// TIA Portal V17 export
// export: Created 2024-08-26T21:07:14.5567643Z, ExportSetting WithDefaults, DisplayName Totally Integrated Automation Portal, DisplayVersion V17 Update 7, DisplayName TIA Portal Openness, DisplayVersion V17 Update 7, DisplayName TIA Portal Version Control Interface, DisplayVersion V17, DisplayName SINAMICS Startdrive Advanced, DisplayVersion V17 SP2, DisplayName SINAMICS Startdrive G110M, G120, G120C, G120D, G120P, G115D, DisplayVersion V17 SP2, DisplayName SINAMICS Startdrive G130, G150, S120, S150, SINAMICS MV, S210, DisplayVersion V17 SP2, DisplayName STEP 7 Professional, DisplayVersion V17 Update 7, DisplayName STEP 7 Safety, DisplayVersion V17 Update 6, DisplayName WinCC Advanced / Unified PC, DisplayVersion V17 Update 7
ORGANIZATION_BLOCK "Main"   // OB1, LAD, ProgramCycle
TITLE = "Main Program Sweep (Cycle)"
{ S7_Optimized_Access := 'TRUE' }
VERSION : 0.1
// stored: AutoNumber true, IsIECCheckEnabled false, SetENOAutomatically false
   VAR_INPUT
      Initial_Call : Bool;   // Initial call of this OB
      Remanence : Bool;   // =True, if remanent data are available
   END_VAR
   VAR_TEMP
      BUFFER : String;
   END_VAR
   VAR_TEMP   // added for the SCL form of the ladder/FBD networks
      _w1 : Bool;
      _w2 : Bool;
      _w3 : Bool;
      _w4 : Bool;
      _w5 : Bool;
      _w6 : Bool;
      _w7 : Bool;
      _w8 : Bool;
      _w9 : Bool;
      _w10 : Bool;
      _w11 : Bool;
   END_VAR
BEGIN

REGION Network 1: SECUENCIA PARA ALARMAR LA MÁQUINA SI SE APAGA A LA MITAD DE UN CICLO DE PRODUCCIÓN
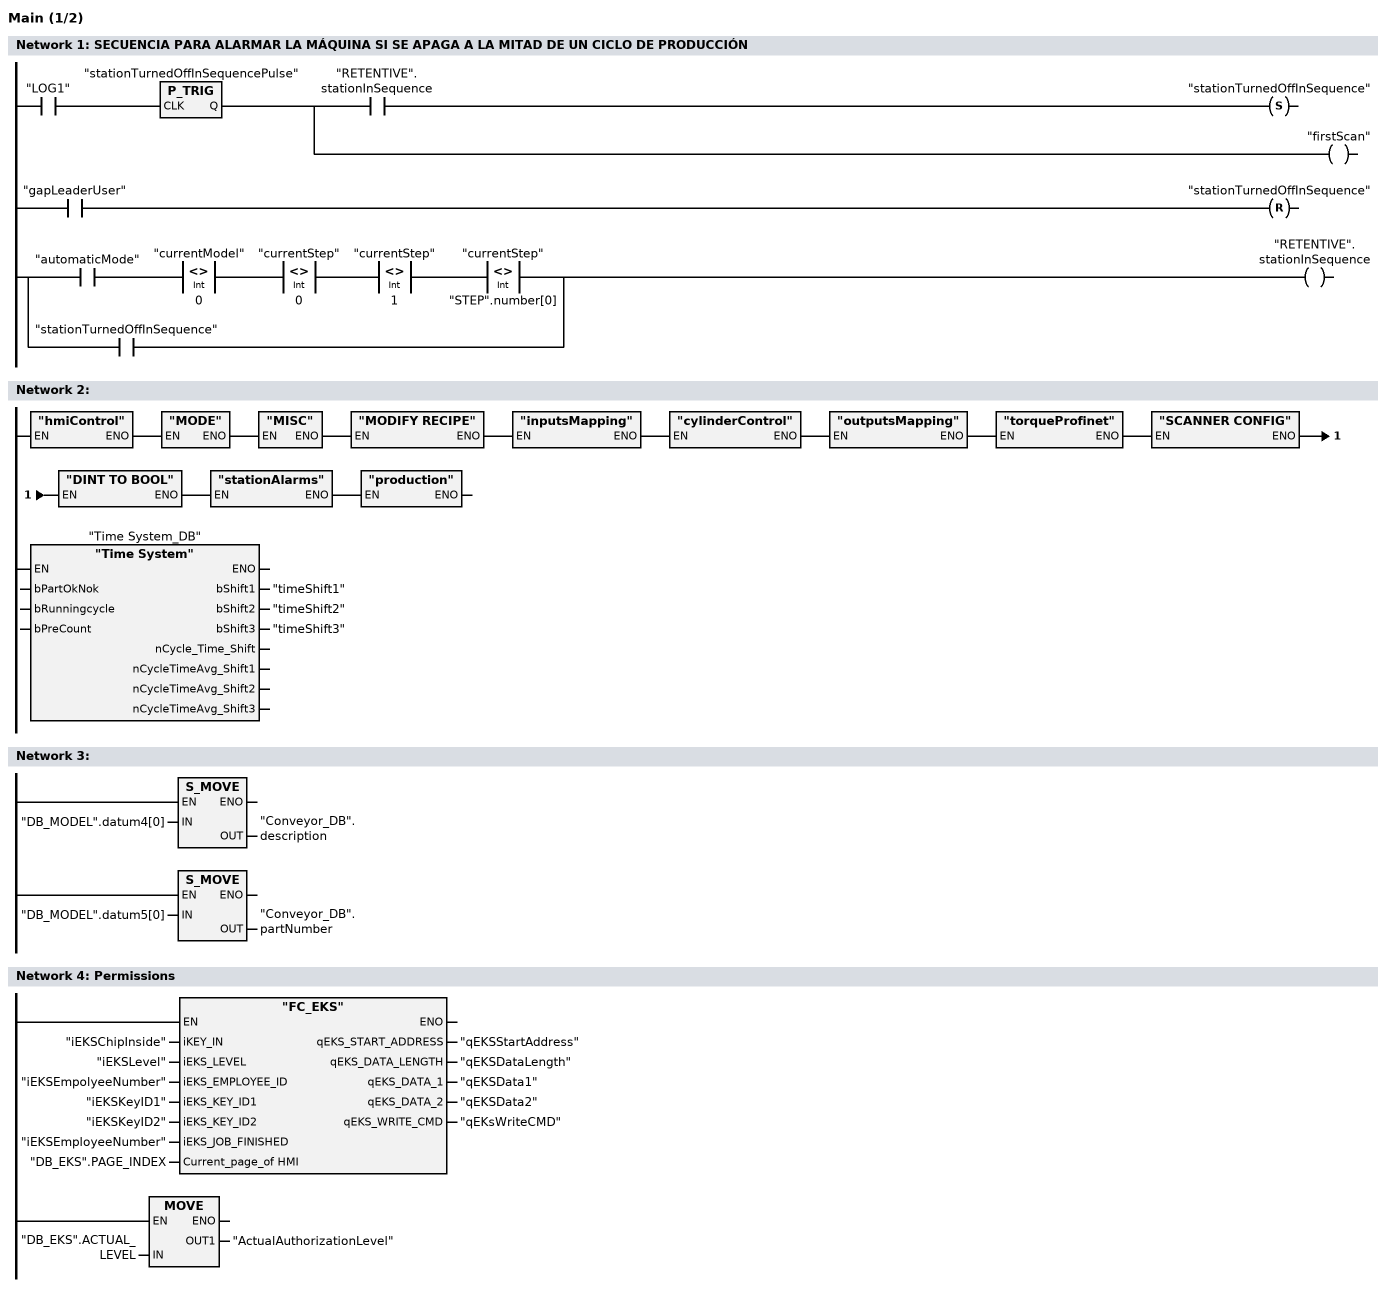
   RUNG wire#powerrail
      Contact( "LOG1" )
      P_Trig( "stationTurnedOffInSequencePulse" )
      wire#w1
      Contact( "RETENTIVE".stationInSequence )
      S_Coil( "stationTurnedOffInSequence" )
   END_RUNG
   RUNG wire#w1
      Coil( "firstScan" )
   END_RUNG
   RUNG wire#powerrail
      Contact( "gapLeaderUser" )
      R_Coil( "stationTurnedOffInSequence" )
   END_RUNG
   RUNG wire#powerrail
      Contact( "automaticMode" )
      { S7_Templates := "SrcType := Int" } NE_Contact(in1 := "currentModel", in2 := 0)
      { S7_Templates := "SrcType := Int" } NE_Contact(in1 := "currentStep", in2 := 0)
      { S7_Templates := "SrcType := Int" } NE_Contact(in1 := "currentStep", in2 := 1)
      { S7_Templates := "SrcType := Int" } NE_Contact(in1 := "currentStep", in2 := "STEP".number[0])
      wire#w2
      Coil( "RETENTIVE".stationInSequence )
   END_RUNG
   RUNG wire#powerrail
      Contact( "stationTurnedOffInSequence" )
   END_RUNG wire#w2
   // the same network as SCL:
   #_w1 := "LOG1" AND NOT "stationTurnedOffInSequencePulse";   // rising edge
   "stationTurnedOffInSequencePulse" := "LOG1";
   IF #_w1 AND "RETENTIVE".stationInSequence THEN "stationTurnedOffInSequence" := TRUE; END_IF;
   "firstScan" := #_w1;
   IF "gapLeaderUser" THEN "stationTurnedOffInSequence" := FALSE; END_IF;
   "RETENTIVE".stationInSequence := ("automaticMode" AND ("currentModel" <> 0) AND ("currentStep" <> 0) AND ("currentStep" <> 1) AND ("currentStep" <> "STEP".number[0])) OR "stationTurnedOffInSequence";
END_REGION

REGION Network 2
   RUNG wire#powerrail
      "hmiControl"()
      "MODE"()
      "MISC"()
      "MODIFY RECIPE"()
      "inputsMapping"()
      "cylinderControl"()
      "outputsMapping"()
      "torqueProfinet"()
      "SCANNER CONFIG"()
      "DINT TO BOOL"()
      "stationAlarms"()
      "production"()
   END_RUNG
   RUNG wire#powerrail
      "Time System_DB"(bPartOkNok :=, bRunningcycle :=, bPreCount :=, bShift1 => "timeShift1", bShift2 => "timeShift2", bShift3 => "timeShift3", nCycle_Time_Shift =>, nCycleTimeAvg_Shift1 =>, nCycleTimeAvg_Shift2 =>, nCycleTimeAvg_Shift3 =>)
   END_RUNG
   // the same network as SCL:
   "hmiControl"(ENO => #_w1);
   "MODE"(EN := #_w1, ENO => #_w2);
   "MISC"(EN := #_w2, ENO => #_w3);
   "MODIFY RECIPE"(EN := #_w3, ENO => #_w4);
   "inputsMapping"(EN := #_w4, ENO => #_w5);
   "cylinderControl"(EN := #_w5, ENO => #_w6);
   "outputsMapping"(EN := #_w6, ENO => #_w7);
   "torqueProfinet"(EN := #_w7, ENO => #_w8);
   "SCANNER CONFIG"(EN := #_w8, ENO => #_w9);
   "DINT TO BOOL"(EN := #_w9, ENO => #_w10);
   "stationAlarms"(EN := #_w10, ENO => #_w11);
   IF #_w11 THEN "production"(); END_IF;
   "Time System_DB"(bShift1 => "timeShift1", bShift2 => "timeShift2", bShift3 => "timeShift3");   // "Time System"
END_REGION

REGION Network 3
   RUNG wire#powerrail
      S_Move(in := "DB_MODEL".datum4[0], out => "Conveyor_DB".description)
   END_RUNG
   RUNG wire#powerrail
      S_Move(in := "DB_MODEL".datum5[0], out => "Conveyor_DB".partNumber)
   END_RUNG
   // the same network as SCL:
   "Conveyor_DB".description := "DB_MODEL".datum4[0];
   "Conveyor_DB".partNumber := "DB_MODEL".datum5[0];
END_REGION

REGION Network 4: Permissions
   RUNG wire#powerrail
      "FC_EKS"(iKEY_IN := "iEKSChipInside", iEKS_LEVEL := "iEKSLevel", iEKS_EMPLOYEE_ID := "iEKSEmpolyeeNumber", iEKS_KEY_ID1 := "iEKSKeyID1", iEKS_KEY_ID2 := "iEKSKeyID2", iEKS_JOB_FINISHED := "iEKSEmployeeNumber", "Current_page_of HMI" := "DB_EKS".PAGE_INDEX, qEKS_START_ADDRESS => "qEKSStartAddress", qEKS_DATA_LENGTH => "qEKSDataLength", qEKS_DATA_1 => "qEKSData1", qEKS_DATA_2 => "qEKSData2", qEKS_WRITE_CMD => "qEKsWriteCMD")
   END_RUNG
   RUNG wire#powerrail
      Move(in := "DB_EKS".ACTUAL_LEVEL, out1 => "ActualAuthorizationLevel")
   END_RUNG
   // the same network as SCL:
   "FC_EKS"(iKEY_IN := "iEKSChipInside",
            iEKS_LEVEL := "iEKSLevel",
            iEKS_EMPLOYEE_ID := "iEKSEmpolyeeNumber",
            iEKS_KEY_ID1 := "iEKSKeyID1",
            iEKS_KEY_ID2 := "iEKSKeyID2",
            iEKS_JOB_FINISHED := "iEKSEmployeeNumber",
            "Current_page_of HMI" := "DB_EKS".PAGE_INDEX,
            qEKS_START_ADDRESS => "qEKSStartAddress",
            qEKS_DATA_LENGTH => "qEKSDataLength",
            qEKS_DATA_1 => "qEKSData1",
            qEKS_DATA_2 => "qEKSData2",
            qEKS_WRITE_CMD => "qEKsWriteCMD");
   "ActualAuthorizationLevel" := "DB_EKS".ACTUAL_LEVEL;
END_REGION

REGION Network 5: Awake signal
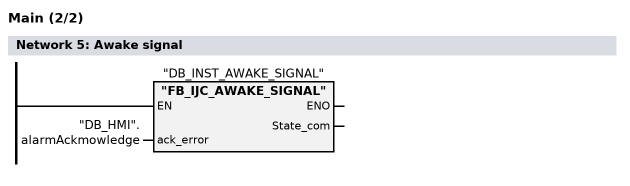
   RUNG wire#powerrail
      "DB_INST_AWAKE_SIGNAL"(ack_error := "DB_HMI".alarmAckmowledge, State_com =>)
   END_RUNG
   // the same network as SCL:
   "DB_INST_AWAKE_SIGNAL"(ack_error := "DB_HMI".alarmAckmowledge);   // "FB_IJC_AWAKE_SIGNAL"
END_REGION
END_ORGANIZATION_BLOCK
